// TIA Portal V18 export
FUNCTION_BLOCK "encoder_mes_speed"   // FB20, FBD
{ S7_Optimized_Access := 'TRUE' }
VERSION : 0.1
// stored: AutoNumber true, IsIECCheckEnabled false, IsRetainMemResEnabled false, MemoryReserve 100, SetENOAutomatically false, UDAEnableTagReadback false
   VAR_INPUT
      Cycle_Time_s : Real;
      Pos : Real;
   END_VAR
   VAR_OUTPUT
      Speed_mm_p_sec : Real;
   END_VAR
   VAR
      MEM : LReal;
      RET_VAL : LReal;
      Pos_was : Real;
   END_VAR
   VAR_TEMP
      Speed_mm_p_sec_temp : Real;
      delta : Real;
      n : Real;
   END_VAR
BEGIN

REGION Network 1
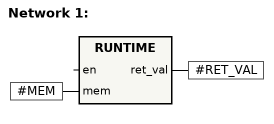
   // no SCL statement known for Runtime: written as a call
   #RET_VAL := Runtime(mem := #MEM);
END_REGION

REGION Network 2 (SCL)
   #delta := #Pos - #Pos_was;
   #Speed_mm_p_sec_temp := #delta / #Cycle_Time_s;
   #n := 10;
   #Speed_mm_p_sec := (#Speed_mm_p_sec * (#n - 1) + #Speed_mm_p_sec_temp)/ #n;

   #Pos_was := #Pos;
END_REGION
END_FUNCTION_BLOCK
